FUNCTION_BLOCK MovingAverage (* moving average filter *)
  (* Standard: 61499-2 *)
  (* Version 1.0, 2026-04-20, Thomas Mayr *)
  PACKAGE eclipse4diac::signalprocessing;
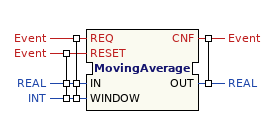
  EVENT_INPUT
    REQ WITH IN, WINDOW; (* Calculate next output *)
    RESET WITH IN, WINDOW; (* Reset internal filter state *)
  END_EVENT
  EVENT_OUTPUT
    CNF WITH OUT; (* Output value updated *)
  END_EVENT
  VAR_INPUT
    IN : REAL; (* Input value *)
    WINDOW : INT; (* Window size (number of samples) *)
  END_VAR
  VAR_OUTPUT
    OUT : REAL; (* Filtered output value *)
  END_VAR
  VAR
    count : INT;
    sum : REAL;
    index : INT;
    buffer : ARRAY [0..99] OF REAL;
    effectiveWindow : INT;
    lastWindow : INT;
    i : INT;
  END_VAR
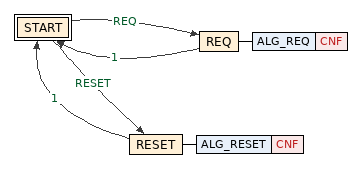
  EC_STATES
    START; (* Initial State *)
    REQ : ALG_REQ -> CNF;
    RESET : ALG_RESET -> CNF;
  END_STATES
  EC_TRANSITIONS
    START TO REQ := REQ;
    REQ TO START := 1;
    START TO RESET := RESET;
    RESET TO START := 1;
  END_TRANSITIONS
  ALGORITHM ALG_REQ IN ST:
IF WINDOW <= 0 THEN
	OUT := IN;
	RETURN;
END_IF;

effectiveWindow := WINDOW;
IF effectiveWindow > 100 THEN
	effectiveWindow := 100;
END_IF;

IF effectiveWindow <> lastWindow THEN
	sum := 0.0;
	index := 0;
	count := 0;
	i := 0;
	WHILE i < 100 DO
		buffer[i] := 0.0;
		i := i + 1;
	END_WHILE;
	lastWindow := effectiveWindow;
END_IF;

IF count < effectiveWindow THEN
	buffer[index] := IN;
	sum := sum + IN;
	count := count + 1;
ELSE
	sum := sum - buffer[index];
	buffer[index] := IN;
	sum := sum + IN;
END_IF;

index := (index + 1) MOD effectiveWindow;

OUT := sum / INT_TO_REAL(count);
  END_ALGORITHM
  ALGORITHM ALG_RESET IN ST:
sum := 0.0;
index := 0;
count := 0;
lastWindow := 0;
i := 0;
WHILE i < 100 DO
	buffer[i] := 0.0;
	i := i + 1;
END_WHILE;
OUT := 0.0;
  END_ALGORITHM
END_FUNCTION_BLOCK
